PROGRAM Bumper
VAR
	BumperStatus		AT%I* : BOOL;
	
	Timer:TOF;
	Timer_Time: TIME := T#5000MS;	
END_VAR

Timer.PT:= Timer_Time;
Timer.IN := BumperStatus;

IF Timer.Q THEN 
	Main.SetBumperaktiv(TRUE);
ELSE
	Main.SetBumperaktiv(FALSE);
END_IF
Timer();

END_PROGRAM

(* stored: Version 1.1.0.1, ProductVersion 3.1.4024.11
   POU Bumper: Id {6efbcee7-f5ea-42a6-97fd-2cdfadcc5d33}, SpecialFunc None *)
